(* IEC 61131-3 sources: AXOpen/src/showcase/app/src/components.keyence.vision/Documentation, 4 files *)

(* ---- Axo_IV3_Showcase.st ---- *)
USING AXOpen.Core;
NAMESPACE AXOpen.Components.Keyence.Vision
    {S7.extern=ReadWrite}
    CLASS Axo_IV3_Showcase EXTENDS AXOpen.Core.AxoObject
        //<ComponentDeclaration>
        VAR PUBLIC
            {#ix-set:DeviceIpAddress = "192.168.1.106"} // Needed for live view
            Component : AXOpen.Components.Keyence.Vision.Axo_IV3;
        END_VAR
        //</ComponentDeclaration>

        //<InitializationArgumentsDeclaration>
        VAR PUBLIC
            {#ix-set:AttributeName = "<#Activate manual control#>"}
            ActivateManualControl : BOOL;
        END_VAR
        //</InitializationArgumentsDeclaration>

        METHOD PUBLIC OVERRIDE Run
            VAR_INPUT
                inParent : IAxoObject;
            END_VAR

            SUPER.Run(inParent);

            IF ActivateManualControl THEN
                Component.ActivateManualControl();
            END_IF;

            //<Initialization>
            Component.Run(      inParent                                          :=   THIS,
                                hwID                                            :=   AXOpen.Showcase.HwIdentifiers#keyence_iv3_HwID);
            //</Initialization>

            THIS.UseInSequencer();
        END_METHOD

        //<Usage>
        VAR PUBLIC
            Sequencer : AxoSequencer;
            Steps : ARRAY[0..3] OF AXOpen.Core.AxoStep;
        END_VAR

        VAR PRIVATE
            _OverAllResult  : BOOL;
            _ResultData  :  ARRAY[0..20] OF UINT;
        END_VAR

        METHOD PRIVATE UseInSequencer

            Sequencer.Run(THIS);
            Sequencer.Open();
            Sequencer.SequenceMode := eAxoSequenceMode#RunOnce;

            IF(Steps[0].Execute(Sequencer, 'Restore')) THEN
                Component.Config.InfoTime    := LTIME#5S;
                Component.Config.ErrorTime   := LTIME#10S;
                Component.Config.TaskTimeout := LTIME#50S;
                Component.Restore();
                Sequencer.MoveNext();
            END_IF;

            IF(Steps[1].Execute(Sequencer, 'Change program')) THEN
                IF(Component.ChangeProgram(UINT#0).IsDone()) THEN
                    Sequencer.MoveNext();
                END_IF;
            END_IF;

            IF(Steps[2].Execute(Sequencer, 'Trigger')) THEN
                IF(Component.Trigger().IsDone()) THEN
                    Sequencer.MoveNext();
                END_IF;
            END_IF;

            IF(Steps[3].Execute(Sequencer, 'Access the result data')) THEN
                _OverAllResult := Component.Inputs.DeviceResultBits_1.OverallJudgmentOK;
                // The meaning of the result data changes with the type of the control,
                // so it must be evaluated individually in the production code
                _ResultData[0] := Component.Inputs.ToolResult_1.MatchingRate;
                _ResultData[1] := Component.Inputs.ToolResult_1.MatchingRateMAX;
                _ResultData[2] := Component.Inputs.ToolResult_1.MatchingRateMIN;
                _ResultData[3] := Component.Inputs.ToolResult_1.LowerThreshold;
                _ResultData[4] := Component.Inputs.ToolResult_1.UpperThreshold;
                _ResultData[5] := Component.Inputs.ToolResult_1.DecimalPointPosition;
                _ResultData[6] := Component.Inputs.ToolResult_1.Data_1;
                _ResultData[7] := Component.Inputs.ToolResult_1.Data_2;
                _ResultData[8] := Component.Inputs.ToolResult_1.Data_3;
                Sequencer.CompleteSequence();
            END_IF;

        END_METHOD
        //</Usage>
    END_CLASS
END_NAMESPACE

(* ---- Axo_SR_1000_Showcase.st ---- *)
USING AXOpen.Core;
NAMESPACE AXOpen.Components.Keyence.Vision
    {S7.extern=ReadWrite}
    CLASS Axo_SR_1000_Showcase EXTENDS AXOpen.Core.AxoObject
        //<ComponentDeclaration>
        VAR PUBLIC
            Component : AXOpen.Components.Keyence.Vision.Axo_SR_1000;
        END_VAR
        //</ComponentDeclaration>

        //<InitializationArgumentsDeclaration>
        VAR PUBLIC
            {#ix-set:AttributeName = "<#Activate manual control#>"}
            ActivateManualControl : BOOL;
        END_VAR
        //</InitializationArgumentsDeclaration>

        METHOD PUBLIC OVERRIDE Run
            VAR_INPUT
                inParent : IAxoObject;
            END_VAR

            SUPER.Run(inParent);

            IF ActivateManualControl THEN
                Component.ActivateManualControl();
            END_IF;

            //<Initialization>
            Component.Run(      inParent                                          :=   THIS,
                                hwID                                            :=   AXOpen.Showcase.HwIdentifiers#keyence_sr_1000_HwID);
            //</Initialization>

            THIS.UseInSequencer();
        END_METHOD

        //<Usage>
        VAR PUBLIC
            Sequencer : AxoSequencer;
            Steps : ARRAY[0..3] OF AXOpen.Core.AxoStep;
        END_VAR

        VAR PRIVATE
            _ResultData  :   AXOpen.Components.Keyence.Vision.Axo_SR_1000_ResultData;
        END_VAR

        METHOD PRIVATE UseInSequencer

            Sequencer.Run(THIS);
            Sequencer.Open();

            IF(Steps[0].Execute(Sequencer, 'Clear result data')) THEN
                IF(Component.ClearResultData().IsDone()) THEN
                    Sequencer.MoveNext();
                END_IF;
            END_IF;

            IF(Steps[1].Execute(Sequencer, 'Tune')) THEN
                IF(Component.Tune(UINT#0).IsDone()) THEN
                    Sequencer.MoveNext();
                END_IF;
            END_IF;

            IF(Steps[2].Execute(Sequencer, 'Read data')) THEN
                IF(Component.Read(UINT#0).IsDone()) THEN
                    Sequencer.MoveNext();
                END_IF;
            END_IF;

            IF(Steps[3].Execute(Sequencer, 'Evaluate data')) THEN
                _ResultData := Component.ResultData;
                Sequencer.CompleteSequence();
            END_IF;

        END_METHOD
        //</Usage>
    END_CLASS
END_NAMESPACE

(* ---- Axo_SR_750_Showcase.st ---- *)
USING AXOpen.Core;
NAMESPACE AXOpen.Components.Keyence.Vision
    {S7.extern=ReadWrite}
    CLASS Axo_SR_750_Showcase EXTENDS AXOpen.Core.AxoObject
        //<ComponentDeclaration>
        VAR PUBLIC
            Component : AXOpen.Components.Keyence.Vision.Axo_SR_750;
        END_VAR
        //</ComponentDeclaration>

        //<InitializationArgumentsDeclaration>
        VAR PUBLIC
            {#ix-set:AttributeName = "<#Activate manual control#>"}
            ActivateManualControl : BOOL;
        END_VAR
        //</InitializationArgumentsDeclaration>

        METHOD PUBLIC OVERRIDE Run
            VAR_INPUT
                inParent : IAxoObject;
            END_VAR

            SUPER.Run(inParent);

            IF ActivateManualControl THEN
                Component.ActivateManualControl();
            END_IF;

            //<Initialization>
            Component.Run(
                                inParent                                          :=   THIS,
                                hwID                                            :=   AXOpen.Showcase.HwIdentifiers#keyence_sr_750_HwID);
            //</Initialization>

            THIS.UseInSequencer();
        END_METHOD

        //<Usage>
        VAR PUBLIC
            Sequencer : AxoSequencer;
            Steps : ARRAY[0..4] OF AXOpen.Core.AxoStep;
        END_VAR

        VAR PRIVATE
            _ResultData  :   AXOpen.Components.Keyence.Vision.Axo_SR_750_ResultData;
        END_VAR

        METHOD PRIVATE UseInSequencer

            Sequencer.Run(THIS);
            Sequencer.Open();
            Sequencer.SequenceMode := eAxoSequenceMode#RunOnce;

            IF(Steps[0].Execute(Sequencer, 'Restore')) THEN
                Component.Config.InfoTime    := LTIME#2S;
                Component.Config.ErrorTime   := LTIME#5S;
                Component.Config.TaskTimeout := LTIME#50S;
                Component.Restore();
                Sequencer.MoveNext();
            END_IF;

            IF(Steps[1].Execute(Sequencer, 'Clear result data')) THEN
                IF(Component.ClearResultData().IsDone()) THEN
                    Sequencer.MoveNext();
                END_IF;
            END_IF;

            IF(Steps[2].Execute(Sequencer, 'Tune')) THEN
                IF(Component.Tune(UINT#0).IsDone()) THEN
                    Sequencer.MoveNext();
                END_IF;
            END_IF;

            IF(Steps[3].Execute(Sequencer, 'Read data')) THEN
                IF(Component.Read(UINT#0).IsDone()) THEN
                    Sequencer.MoveNext();
                END_IF;
            END_IF;

            IF(Steps[4].Execute(Sequencer, 'Evaluate data')) THEN
                _ResultData := Component.ResultData;
                Sequencer.CompleteSequence();
            END_IF;

        END_METHOD
        //</Usage>
    END_CLASS
END_NAMESPACE

(* ---- KeyenceVision.st ---- *)
NAMESPACE AXOpen.Components.Keyence.Vision
    {S7.extern=ReadWrite}
    CLASS KeyenceVision EXTENDS AXOpen.Core.AxoObject
        VAR PUBLIC
            rootObject      : AxoObject;
            axo_SR_750    : AXOpen.Components.Keyence.Vision.Axo_SR_750_Showcase;
            axo_SR_1000    : AXOpen.Components.Keyence.Vision.Axo_SR_1000_Showcase;
            axo_IV3  : AXOpen.Components.Keyence.Vision.Axo_IV3_Showcase;
        END_VAR

        METHOD PUBLIC Execute
            rootObject.Run(THIS);
            axo_SR_750.Run(rootObject);
            axo_SR_1000.Run(rootObject);
            axo_IV3.Run(rootObject);
        END_METHOD
    END_CLASS
END_NAMESPACE
